ABB RAPID module: Module1.mod

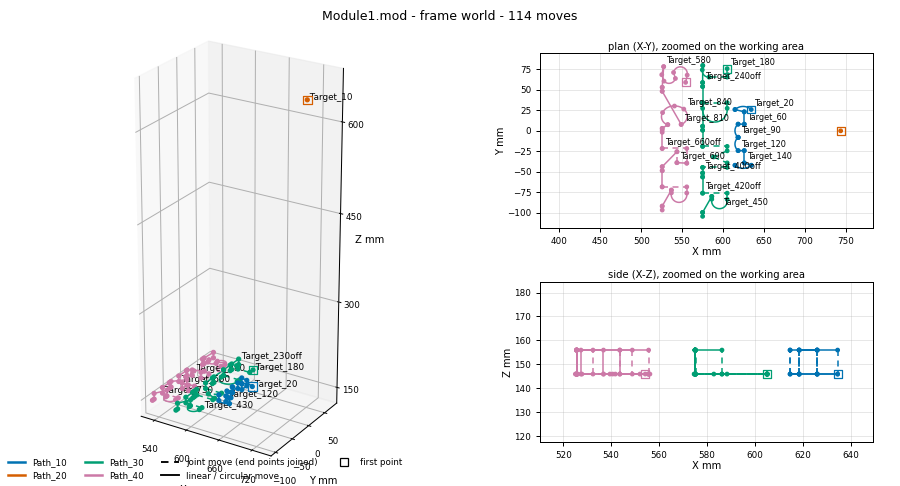
[picture p0: tool path of Module1.mod in frame world, 114 of 114 moves have a stored position in this frame; points joined in program order, loops and branches not executed]
MODULE Module1
    CONST robtarget Target_20:=[[25.588,146.054,0],[1,0,0,0],[0,0,0,1],[9E+09,9E+09,9E+09,9E+09,9E+09,9E+09]];
    CONST robtarget Target_30:=[[35.494,149.81,0],[1,0,0,0],[0,0,0,1],[9E+09,9E+09,9E+09,9E+09,9E+09,9E+09]];
    CONST robtarget Target_Home:=[[306.283094642,150.004,-445.953252285],[1,0,0.000000007,0],[0,0,0,1],[9E+09,9E+09,9E+09,9E+09,9E+09,9E+09]];
    CONST robtarget Target_10:=[[-83.715981405,120.000002402,-514.953287941],[1,-0.000000013,-0.000000023,0.000000007],[-1,0,0,0],[9E+09,9E+09,9E+09,9E+09,9E+09,9E+09]];
    CONST robtarget Target_40:=[[45.401,146.054,0],[1,0,0,0],[0,0,0,1],[9E+09,9E+09,9E+09,9E+09,9E+09,9E+09]];
    CONST robtarget Target_40off:=[[45.401,146.054,-10],[1,0,0,0],[0,0,0,1],[9E+09,9E+09,9E+09,9E+09,9E+09,9E+09]];
    CONST robtarget Target_50:=[[34.121,143.221,0],[1,0,0,0],[0,0,0,1],[9E+09,9E+09,9E+09,9E+09,9E+09,9E+09]];
    CONST robtarget Target_50off:=[[34.121,143.221,-10],[1,0,0,0],[0,0,0,1],[9E+09,9E+09,9E+09,9E+09,9E+09,9E+09]];
    CONST robtarget Target_60:=[[34.121,128.148,0],[1,0,0,0],[0,0,0,1],[9E+09,9E+09,9E+09,9E+09,9E+09,9E+09]];
    CONST robtarget Target_60off:=[[34.121,128.148,-10],[1,0,0,0],[0,0,0,1],[9E+09,9E+09,9E+09,9E+09,9E+09,9E+09]];
    CONST robtarget Target_70:=[[41.621,128.173,0],[1,0,0,0],[0,0,0,1],[9E+09,9E+09,9E+09,9E+09,9E+09,9E+09]];
    CONST robtarget Target_70off:=[[41.621,128.173,-10],[1,0,0,0],[0,0,0,1],[9E+09,9E+09,9E+09,9E+09,9E+09,9E+09]];
    CONST robtarget Target_80:=[[45.462,120.186,0],[1,0,0,0],[0,0,0,1],[9E+09,9E+09,9E+09,9E+09,9E+09,9E+09]];
    CONST robtarget Target_90:=[[41.621,112.188,0],[1,0,0,0],[0,0,0,1],[9E+09,9E+09,9E+09,9E+09,9E+09,9E+09]];
    CONST robtarget Target_90off:=[[41.621,112.188,-10],[1,0,0,0],[0,0,0,1],[9E+09,9E+09,9E+09,9E+09,9E+09,9E+09]];
    CONST robtarget Target_110:=[[45.462,103.801,0],[1,0,0,0],[0,0,0,1],[9E+09,9E+09,9E+09,9E+09,9E+09,9E+09]];
    CONST robtarget Target_110off:=[[45.462,103.801,-10],[1,0,0,0],[0,0,0,1],[9E+09,9E+09,9E+09,9E+09,9E+09,9E+09]];
    CONST robtarget Target_120:=[[41.621,95.802,0],[1,0,0,0],[0,0,0,1],[9E+09,9E+09,9E+09,9E+09,9E+09,9E+09]];
    CONST robtarget Target_120off:=[[41.621,95.802,-10],[1,0,0,0],[0,0,0,1],[9E+09,9E+09,9E+09,9E+09,9E+09,9E+09]];
    CONST robtarget Target_130:=[[34.121,95.839,0],[1,0,0,0],[0,0,0,1],[9E+09,9E+09,9E+09,9E+09,9E+09,9E+09]];
    CONST robtarget Target_130off:=[[34.121,95.839,-10],[1,0,0,0],[0,0,0,1],[9E+09,9E+09,9E+09,9E+09,9E+09,9E+09]];
    CONST robtarget Target_140:=[[34.121,80.766,0],[1,0,0,0],[0,0,0,1],[9E+09,9E+09,9E+09,9E+09,9E+09,9E+09]];
    CONST robtarget Target_140off:=[[34.121,80.766,-10],[1,0,0,0],[0,0,0,1],[9E+09,9E+09,9E+09,9E+09,9E+09,9E+09]];
    CONST robtarget Target_150:=[[25.588,77.934,0],[1,0,0,0],[0,0,0,1],[9E+09,9E+09,9E+09,9E+09,9E+09,9E+09]];
    CONST robtarget Target_150off:=[[25.588,77.934,-10],[1,0,0,0],[0,0,0,1],[9E+09,9E+09,9E+09,9E+09,9E+09,9E+09]];
    CONST robtarget Target_160:=[[35.494,74.178,0],[1,0,0,0],[0,0,0,1],[9E+09,9E+09,9E+09,9E+09,9E+09,9E+09]];
    CONST robtarget Target_170:=[[45.401,77.934,0],[1,0,0,0],[0,0,0,1],[9E+09,9E+09,9E+09,9E+09,9E+09,9E+09]];
    CONST robtarget Target_170off:=[[45.401,77.934,-10],[1,0,0,0],[0,0,0,1],[9E+09,9E+09,9E+09,9E+09,9E+09,9E+09]];
    CONST robtarget Target_100:=[[41.621,111.787,0],[1,0,0,0],[0,0,0,1],[9E+09,9E+09,9E+09,9E+09,9E+09,9E+09]];
    CONST robtarget Target_100off:=[[41.621,111.787,-10],[1,0,0,0],[0,0,0,1],[9E+09,9E+09,9E+09,9E+09,9E+09,9E+09]];
    CONST robtarget Target_180:=[[55,195.989,0],[1,0,0,0],[0,0,0,1],[9E+09,9E+09,9E+09,9E+09,9E+09,9E+09]];
    CONST robtarget Target_190:=[[55,185.656,0],[1,0,0,0],[0,0,0,1],[9E+09,9E+09,9E+09,9E+09,9E+09,9E+09]];
    CONST robtarget Target_200:=[[77.196,185.656,0],[1,0,0,0],[0,0,0,1],[9E+09,9E+09,9E+09,9E+09,9E+09,9E+09]];
    CONST robtarget Target_210:=[[83.274,188.063,0],[1,0,0,0],[0,0,0,1],[9E+09,9E+09,9E+09,9E+09,9E+09,9E+09]];
    CONST robtarget Target_220:=[[85.413,194.53,0],[1,0,0,0],[0,0,0,1],[9E+09,9E+09,9E+09,9E+09,9E+09,9E+09]];
    CONST robtarget Target_230:=[[84.83,199.83,0],[1,0,0,0],[0,0,0,1],[9E+09,9E+09,9E+09,9E+09,9E+09,9E+09]];
    CONST robtarget Target_240:=[[85,178.995,0],[1,0,0,0],[0,0,0,1],[9E+09,9E+09,9E+09,9E+09,9E+09,9E+09]];
    CONST robtarget Target_230off:=[[84.83,199.83,-10],[1,0,0,0],[0,0,0,1],[9E+09,9E+09,9E+09,9E+09,9E+09,9E+09]];
    CONST robtarget Target_240off:=[[85,178.995,-10],[1,0,0,0],[0,0,0,1],[9E+09,9E+09,9E+09,9E+09,9E+09,9E+09]];
    CONST robtarget Target_250:=[[85,174.182,0],[1,0,0,0],[0,0,0,1],[9E+09,9E+09,9E+09,9E+09,9E+09,9E+09]];
    CONST robtarget Target_260:=[[55,154.392,0],[1,0,0,0],[0,0,0,1],[9E+09,9E+09,9E+09,9E+09,9E+09,9E+09]];
    CONST robtarget Target_250off:=[[85,174.182,-10],[1,0,0,0],[0,0,0,1],[9E+09,9E+09,9E+09,9E+09,9E+09,9E+09]];
    CONST robtarget Target_260off:=[[55,154.392,-10],[1,0,0,0],[0,0,0,1],[9E+09,9E+09,9E+09,9E+09,9E+09,9E+09]];
    CONST robtarget Target_270:=[[55,147.561,0],[1,0,0,0],[0,0,0,1],[9E+09,9E+09,9E+09,9E+09,9E+09,9E+09]];
    CONST robtarget Target_280:=[[70.024,130.737,0],[1,0,0,0],[0,0,0,1],[9E+09,9E+09,9E+09,9E+09,9E+09,9E+09]];
    CONST robtarget Target_290:=[[85,147.488,0],[1,0,0,0],[0,0,0,1],[9E+09,9E+09,9E+09,9E+09,9E+09,9E+09]];
    CONST robtarget Target_300:=[[85,154.392,0],[1,0,0,0],[0,0,0,1],[9E+09,9E+09,9E+09,9E+09,9E+09,9E+09]];
    CONST robtarget Target_300off:=[[85,154.392,-10],[1,0,0,0],[0,0,0,1],[9E+09,9E+09,9E+09,9E+09,9E+09,9E+09]];
    CONST robtarget Target_310:=[[85,125.632,0],[1,0,0,0],[0,0,0,1],[9E+09,9E+09,9E+09,9E+09,9E+09,9E+09]];
    CONST robtarget Target_320:=[[85,120.818,0],[1,0,0,0],[0,0,0,1],[9E+09,9E+09,9E+09,9E+09,9E+09,9E+09]];
    CONST robtarget Target_310off:=[[85,125.632,-10],[1,0,0,0],[0,0,0,1],[9E+09,9E+09,9E+09,9E+09,9E+09,9E+09]];
    CONST robtarget Target_320off:=[[85,120.818,-10],[1,0,0,0],[0,0,0,1],[9E+09,9E+09,9E+09,9E+09,9E+09,9E+09]];
    CONST robtarget Target_330:=[[85,101.029,0],[1,0,0,0],[0,0,0,1],[9E+09,9E+09,9E+09,9E+09,9E+09,9E+09]];
    CONST robtarget Target_330off:=[[85,101.029,-10],[1,0,0,0],[0,0,0,1],[9E+09,9E+09,9E+09,9E+09,9E+09,9E+09]];
    CONST robtarget Target_340:=[[55,101.029,0],[1,0,0,0],[0,0,0,1],[9E+09,9E+09,9E+09,9E+09,9E+09,9E+09]];
    CONST robtarget Target_350:=[[55,95.583,0],[1,0,0,0],[0,0,0,1],[9E+09,9E+09,9E+09,9E+09,9E+09,9E+09]];
    CONST robtarget Target_360:=[[71.702,88.096,0],[1,0,0,0],[0,0,0,1],[9E+09,9E+09,9E+09,9E+09,9E+09,9E+09]];
    CONST robtarget Target_370:=[[55,80.851,0],[1,0,0,0],[0,0,0,1],[9E+09,9E+09,9E+09,9E+09,9E+09,9E+09]];
    CONST robtarget Target_380:=[[55,75.308,0],[1,0,0,0],[0,0,0,1],[9E+09,9E+09,9E+09,9E+09,9E+09,9E+09]];
    CONST robtarget Target_390:=[[85,75.308,0],[1,0,0,0],[0,0,0,1],[9E+09,9E+09,9E+09,9E+09,9E+09,9E+09]];
    CONST robtarget Target_390off:=[[85,75.308,-10],[1,0,0,0],[0,0,0,1],[9E+09,9E+09,9E+09,9E+09,9E+09,9E+09]];
    CONST robtarget Target_400:=[[85,68.452,0],[1,0,0,0],[0,0,0,1],[9E+09,9E+09,9E+09,9E+09,9E+09,9E+09]];
    CONST robtarget Target_400off:=[[85,68.452,-10],[1,0,0,0],[0,0,0,1],[9E+09,9E+09,9E+09,9E+09,9E+09,9E+09]];
    CONST robtarget Target_410:=[[85,63.639,0],[1,0,0,0],[0,0,0,1],[9E+09,9E+09,9E+09,9E+09,9E+09,9E+09]];
    CONST robtarget Target_420:=[[85,43.849,0],[1,0,0,0],[0,0,0,1],[9E+09,9E+09,9E+09,9E+09,9E+09,9E+09]];
    CONST robtarget Target_410off:=[[85,63.639,-10],[1,0,0,0],[0,0,0,1],[9E+09,9E+09,9E+09,9E+09,9E+09,9E+09]];
    CONST robtarget Target_420off:=[[85,43.849,-10],[1,0,0,0],[0,0,0,1],[9E+09,9E+09,9E+09,9E+09,9E+09,9E+09]];
    CONST robtarget Target_430:=[[55,43.849,0],[1,0,0,0],[0,0,0,1],[9E+09,9E+09,9E+09,9E+09,9E+09,9E+09]];
    CONST robtarget Target_440:=[[55,36.313,0],[1,0,0,0],[0,0,0,1],[9E+09,9E+09,9E+09,9E+09,9E+09,9E+09]];
    CONST robtarget Target_450:=[[64.044,24.887,0],[1,0,0,0],[0,0,0,1],[9E+09,9E+09,9E+09,9E+09,9E+09,9E+09]];
    CONST robtarget Target_460:=[[73.817,36.483,0],[1,0,0,0],[0,0,0,1],[9E+09,9E+09,9E+09,9E+09,9E+09,9E+09]];
    CONST robtarget Target_470:=[[73.817,39.862,0],[1,0,0,0],[0,0,0,1],[9E+09,9E+09,9E+09,9E+09,9E+09,9E+09]];
    CONST robtarget Target_480:=[[85,20.316,0],[1,0,0,0],[0,0,0,1],[9E+09,9E+09,9E+09,9E+09,9E+09,9E+09]];
    CONST robtarget Target_470off:=[[73.817,39.862,-10],[1,0,0,0],[0,0,0,1],[9E+09,9E+09,9E+09,9E+09,9E+09,9E+09]];
    CONST robtarget Target_480off:=[[85,20.316,-10],[1,0,0,0],[0,0,0,1],[9E+09,9E+09,9E+09,9E+09,9E+09,9E+09]];
    CONST robtarget Target_490:=[[85,15.502,0],[1,0,0,0],[0,0,0,1],[9E+09,9E+09,9E+09,9E+09,9E+09,9E+09]];
    CONST robtarget Target_500:=[[105.804,179.214,0],[1,0,0,0],[0,0,0,1],[9E+09,9E+09,9E+09,9E+09,9E+09,9E+09]];
    CONST robtarget Target_510:=[[103.859,188.136,0],[1,0,0,0],[0,0,0,1],[9E+09,9E+09,9E+09,9E+09,9E+09,9E+09]];
    CONST robtarget Target_520:=[[112.441,198.225,0],[1,0,0,0],[0,0,0,1],[9E+09,9E+09,9E+09,9E+09,9E+09,9E+09]];
    CONST robtarget Target_530:=[[120.513,191.321,0],[1,0,0,0],[0,0,0,1],[9E+09,9E+09,9E+09,9E+09,9E+09,9E+09]];
    CONST robtarget Target_540:=[[118.276,184.003,0],[1,0,0,0],[0,0,0,1],[9E+09,9E+09,9E+09,9E+09,9E+09,9E+09]];
    CONST robtarget Target_550:=[[125.837,178.047,0],[1,0,0,0],[0,0,0,1],[9E+09,9E+09,9E+09,9E+09,9E+09,9E+09]];
    CONST robtarget Target_560:=[[132.206,180.77,0],[1,0,0,0],[0,0,0,1],[9E+09,9E+09,9E+09,9E+09,9E+09,9E+09]];
    CONST robtarget Target_550off:=[[125.837,178.047,-10],[1,0,0,0],[0,0,0,1],[9E+09,9E+09,9E+09,9E+09,9E+09,9E+09]];
    CONST robtarget Target_560off:=[[132.206,180.77,-10],[1,0,0,0],[0,0,0,1],[9E+09,9E+09,9E+09,9E+09,9E+09,9E+09]];
    CONST robtarget Target_570:=[[134.929,188.598,0],[1,0,0,0],[0,0,0,1],[9E+09,9E+09,9E+09,9E+09,9E+09,9E+09]];
    CONST robtarget Target_580:=[[132.595,198.444,0],[1,0,0,0],[0,0,0,1],[9E+09,9E+09,9E+09,9E+09,9E+09,9E+09]];
    CONST robtarget Target_590:=[[134.394,173.209,0],[1,0,0,0],[0,0,0,1],[9E+09,9E+09,9E+09,9E+09,9E+09,9E+09]];
    CONST robtarget Target_600:=[[134.394,168.395,0],[1,0,0,0],[0,0,0,1],[9E+09,9E+09,9E+09,9E+09,9E+09,9E+09]];
    CONST robtarget Target_610:=[[106.388,127.553,0],[1,0,0,0],[0,0,0,1],[9E+09,9E+09,9E+09,9E+09,9E+09,9E+09]];
    CONST robtarget Target_580off:=[[132.595,198.444,-10],[1,0,0,0],[0,0,0,1],[9E+09,9E+09,9E+09,9E+09,9E+09,9E+09]];
    CONST robtarget Target_590off:=[[134.394,173.209,-10],[1,0,0,0],[0,0,0,1],[9E+09,9E+09,9E+09,9E+09,9E+09,9E+09]];
    CONST robtarget Target_600off:=[[134.394,168.395,-10],[1,0,0,0],[0,0,0,1],[9E+09,9E+09,9E+09,9E+09,9E+09,9E+09]];
    CONST robtarget Target_610off:=[[106.388,127.553,-10],[1,0,0,0],[0,0,0,1],[9E+09,9E+09,9E+09,9E+09,9E+09,9E+09]];
    CONST robtarget Target_620:=[[119.419,150.308,0],[1,0,0,0],[0,0,0,1],[9E+09,9E+09,9E+09,9E+09,9E+09,9E+09]];
    CONST robtarget Target_630:=[[132.352,127.553,0],[1,0,0,0],[0,0,0,1],[9E+09,9E+09,9E+09,9E+09,9E+09,9E+09]];
    CONST robtarget Target_640:=[[134.394,123.055,0],[1,0,0,0],[0,0,0,1],[9E+09,9E+09,9E+09,9E+09,9E+09,9E+09]];
    CONST robtarget Target_630off:=[[132.352,127.553,-10],[1,0,0,0],[0,0,0,1],[9E+09,9E+09,9E+09,9E+09,9E+09,9E+09]];
    CONST robtarget Target_640off:=[[134.394,123.055,-10],[1,0,0,0],[0,0,0,1],[9E+09,9E+09,9E+09,9E+09,9E+09,9E+09]];
    CONST robtarget Target_650:=[[134.394,118.241,0],[1,0,0,0],[0,0,0,1],[9E+09,9E+09,9E+09,9E+09,9E+09,9E+09]];
    CONST robtarget Target_660:=[[134.394,98.452,0],[1,0,0,0],[0,0,0,1],[9E+09,9E+09,9E+09,9E+09,9E+09,9E+09]];
    CONST robtarget Target_650off:=[[134.394,120.939,-10],[1,0,0,0],[0,0,0,1],[9E+09,9E+09,9E+09,9E+09,9E+09,9E+09]];
    CONST robtarget Target_660off:=[[134.394,98.452,-10],[1,0,0,0],[0,0,0,1],[9E+09,9E+09,9E+09,9E+09,9E+09,9E+09]];
    CONST robtarget Target_670:=[[104.394,98.452,0],[1,0,0,0],[0,0,0,1],[9E+09,9E+09,9E+09,9E+09,9E+09,9E+09]];
    CONST robtarget Target_680:=[[104.394,80.511,0],[1,0,0,0],[0,0,0,1],[9E+09,9E+09,9E+09,9E+09,9E+09,9E+09]];
    CONST robtarget Target_690:=[[116.404,81.094,0],[1,0,0,0],[0,0,0,1],[9E+09,9E+09,9E+09,9E+09,9E+09,9E+09]];
    CONST robtarget Target_680off:=[[104.394,80.511,-10],[1,0,0,0],[0,0,0,1],[9E+09,9E+09,9E+09,9E+09,9E+09,9E+09]];
    CONST robtarget Target_690off:=[[116.404,81.094,-10],[1,0,0,0],[0,0,0,1],[9E+09,9E+09,9E+09,9E+09,9E+09,9E+09]];
    CONST robtarget Target_700:=[[116.404,94.465,0],[1,0,0,0],[0,0,0,1],[9E+09,9E+09,9E+09,9E+09,9E+09,9E+09]];
    CONST robtarget Target_710:=[[134.394,76.159,0],[1,0,0,0],[0,0,0,1],[9E+09,9E+09,9E+09,9E+09,9E+09,9E+09]];
    CONST robtarget Target_700off:=[[116.404,94.465,-10],[1,0,0,0],[0,0,0,1],[9E+09,9E+09,9E+09,9E+09,9E+09,9E+09]];
    CONST robtarget Target_710off:=[[134.394,76.159,-10],[1,0,0,0],[0,0,0,1],[9E+09,9E+09,9E+09,9E+09,9E+09,9E+09]];
    CONST robtarget Target_720:=[[134.394,71.345,0],[1,0,0,0],[0,0,0,1],[9E+09,9E+09,9E+09,9E+09,9E+09,9E+09]];
    CONST robtarget Target_730:=[[134.394,51.556,0],[1,0,0,0],[0,0,0,1],[9E+09,9E+09,9E+09,9E+09,9E+09,9E+09]];
    CONST robtarget Target_720off:=[[134.394,71.345,-10],[1,0,0,0],[0,0,0,1],[9E+09,9E+09,9E+09,9E+09,9E+09,9E+09]];
    CONST robtarget Target_730off:=[[134.394,51.556,-10],[1,0,0,0],[0,0,0,1],[9E+09,9E+09,9E+09,9E+09,9E+09,9E+09]];
    CONST robtarget Target_740:=[[104.394,51.556,0],[1,0,0,0],[0,0,0,1],[9E+09,9E+09,9E+09,9E+09,9E+09,9E+09]];
    CONST robtarget Target_750:=[[104.394,44.019,0],[1,0,0,0],[0,0,0,1],[9E+09,9E+09,9E+09,9E+09,9E+09,9E+09]];
    CONST robtarget Target_760:=[[113.438,32.593,0],[1,0,0,0],[0,0,0,1],[9E+09,9E+09,9E+09,9E+09,9E+09,9E+09]];
    CONST robtarget Target_770:=[[123.211,44.19,0],[1,0,0,0],[0,0,0,1],[9E+09,9E+09,9E+09,9E+09,9E+09,9E+09]];
    CONST robtarget Target_780:=[[123.211,47.569,0],[1,0,0,0],[0,0,0,1],[9E+09,9E+09,9E+09,9E+09,9E+09,9E+09]];
    CONST robtarget Target_790:=[[134.394,28.023,0],[1,0,0,0],[0,0,0,1],[9E+09,9E+09,9E+09,9E+09,9E+09,9E+09]];
    CONST robtarget Target_780off:=[[123.211,47.569,-10],[1,0,0,0],[0,0,0,1],[9E+09,9E+09,9E+09,9E+09,9E+09,9E+09]];
    CONST robtarget Target_790off:=[[134.394,28.023,-10],[1,0,0,0],[0,0,0,1],[9E+09,9E+09,9E+09,9E+09,9E+09,9E+09]];
    CONST robtarget Target_800:=[[134.394,23.209,0],[1,0,0,0],[0,0,0,1],[9E+09,9E+09,9E+09,9E+09,9E+09,9E+09]];
    CONST robtarget Target_810:=[[111.201,127.869,0],[1,0,0,0],[0,0,0,1],[9E+09,9E+09,9E+09,9E+09,9E+09,9E+09]];
    CONST robtarget Target_820:=[[127.587,127.553,0],[1,0,0,0],[0,0,0,1],[9E+09,9E+09,9E+09,9E+09,9E+09,9E+09]];
    CONST robtarget Target_810off:=[[111.201,127.869,-10],[1,0,0,0],[0,0,0,1],[9E+09,9E+09,9E+09,9E+09,9E+09,9E+09]];
    CONST robtarget Target_820off:=[[127.587,127.553,-10],[1,0,0,0],[0,0,0,1],[9E+09,9E+09,9E+09,9E+09,9E+09,9E+09]];
    CONST robtarget Target_830:=[[103.859,136.815,0],[1,0,0,0],[0,0,0,1],[9E+09,9E+09,9E+09,9E+09,9E+09,9E+09]];
    CONST robtarget Target_840:=[[107.992,146.564,0],[1,0,0,0],[0,0,0,1],[9E+09,9E+09,9E+09,9E+09,9E+09,9E+09]];
    CONST robtarget Target_850:=[[112.855,149.348,0],[1,0,0,0],[0,0,0,1],[9E+09,9E+09,9E+09,9E+09,9E+09,9E+09]];
    CONST robtarget Target_860:=[[119.419,150.308,0],[1,0,0,0],[0,0,0,1],[9E+09,9E+09,9E+09,9E+09,9E+09,9E+09]];
    CONST robtarget Target_870:=[[126.128,149.323,0],[1,0,0,0],[0,0,0,1],[9E+09,9E+09,9E+09,9E+09,9E+09,9E+09]];
    CONST robtarget Target_880:=[[133.944,142.273,0],[1,0,0,0],[0,0,0,1],[9E+09,9E+09,9E+09,9E+09,9E+09,9E+09]];
    CONST robtarget Target_890:=[[134.71,133.971,0],[1,0,0,0],[0,0,0,1],[9E+09,9E+09,9E+09,9E+09,9E+09,9E+09]];
    PERS tooldata MyNewTool:=[TRUE,[[80.603,0,147.485],[0.866025404,0,0.5,0]],[1,[0,0,1],[1,0,0,0],0,0,0]];
    TASK PERS wobjdata Workobject_2:=[FALSE,TRUE,"",[[0,0,0],[1,0,0,0]],[[660,-120,146],[0,0,1,0]]];
    TASK PERS wobjdata Workobject_1:=[FALSE,TRUE,"",[[0,0,0],[1,0,0,0]],[[749.999,-150.004,90],[0,0,1,0]]];

    PROC main()
        Path_20;
        WaitTime 4;
        Path_10;
        Path_20;
        Path_30;
        Path_20;
        Path_40;
        Path_20;
    ENDPROC
    PROC Path_10()                  !Emoji
        MoveJ Target_20,v100,z10,MyNewTool\WObj:=Workobject_2;
        MoveC Target_30, Target_40, v100,z10,MyNewTool\WObj:=Workobject_2;
        WaitTime 1;
        MoveJ Target_40off,v100,z10,MyNewTool\WObj:=Workobject_2;
        MoveL Target_50off,v100,z10,MyNewTool\WObj:=Workobject_2;
        WaitTime 1;
        MoveJ Target_50,v100,z10,MyNewTool\WObj:=Workobject_2;
        MoveL Target_60,v100,z10,MyNewTool\WObj:=Workobject_2;
        WaitTime 1;
        MoveJ Target_60off,v100,z10,MyNewTool\WObj:=Workobject_2;
        MoveL Target_70off,v100,z10,MyNewTool\WObj:=Workobject_2;
        MoveJ Target_70,v100,z10,MyNewTool\WObj:=Workobject_2;
        WaitTime 1;
        MoveC Target_80,Target_90,v100,z10,MyNewTool\WObj:=Workobject_2;
        MoveJ Target_90off,v100,z10,MyNewTool\WObj:=Workobject_2;
        MoveL Target_100off,v100,z10,MyNewTool\WObj:=Workobject_2;
        MoveJ Target_100,v100,z10,MyNewTool\WObj:=Workobject_2;
        WaitTime 1;
        MoveC Target_110,Target_120,v100,z10,MyNewTool\WObj:=Workobject_2;
        MoveJ Target_120off,v100,z100,MyNewTool\WObj:=Workobject_2;
        MoveL Target_130off,v100,z10,MyNewTool\WObj:=Workobject_2;
        MoveJ Target_130,v100,z10,MyNewTool\WObj:=Workobject_2;
        WaitTime 1;
        MoveL Target_140,v100,z10,MyNewTool\WObj:=Workobject_2;
        MoveJ Target_140off,v100,z10,MyNewTool\WObj:=Workobject_2;
        MoveL Target_150off,v100,z10,MyNewTool\WObj:=Workobject_2;
        MoveJ Target_150,v100,z10,MyNewTool\WObj:=Workobject_2;
        MoveC Target_160,Target_170,v100,z10,MyNewTool\WObj:=Workobject_2;
        WaitTime 1;
        MoveJ Target_170off,v100,z10,MyNewTool\WObj:=Workobject_2;
    ENDPROC
    PROC Path_20() !Home
        MoveJ Target_10,v100,z10,MyNewTool\WObj:=Workobject_2;
    ENDPROC
    PROC Path_30() !Iniciales JDMP
        MoveJ Target_180,v100,z10,MyNewTool\WObj:=Workobject_2;    !J
        MoveJ Target_190,v100,z10,MyNewTool\WObj:=Workobject_2;
        MoveJ Target_200,v100,z10,MyNewTool\WObj:=Workobject_2;
        MoveC Target_210,Target_220,v100,z10,MyNewTool\WObj:=Workobject_2;
        MoveJ Target_230,v100,z10,MyNewTool\WObj:=Workobject_2;
        MoveJ Target_230off,v100,z10,MyNewTool\WObj:=Workobject_2;
        MoveL Target_240off,v100,z10,MyNewTool\WObj:=Workobject_2;
        MoveJ Target_240,v100,z10,MyNewTool\WObj:=Workobject_2;
        MoveJ Target_250,v100,z10,MyNewTool\WObj:=Workobject_2;
        MoveJ Target_250off,v100,z10,MyNewTool\WObj:=Workobject_2;
        MoveL Target_300off,v100,z10,MyNewTool\WObj:=Workobject_2; !D
        MoveL Target_300,v100,z10,MyNewTool\WObj:=Workobject_2;
        MoveJ Target_260,v100,z10,MyNewTool\WObj:=Workobject_2;
        MoveL Target_270,v100,z10,MyNewTool\WObj:=Workobject_2;
        MoveC Target_280,Target_290,v100,z10,MyNewTool\WObj:=Workobject_2;
        MoveJ Target_300,v100,z10,MyNewTool\WObj:=Workobject_2;
        MoveL Target_300off,v100,z10,MyNewTool\WObj:=Workobject_2;
        MoveL Target_310off,v100,z10,MyNewTool\WObj:=Workobject_2;
        MoveJ Target_310,v100,z10,MyNewTool\WObj:=Workobject_2;
        MoveJ Target_320,v100,z10,MyNewTool\WObj:=Workobject_2;
        MoveL Target_320off,v100,z10,MyNewTool\WObj:=Workobject_2;
        MoveL Target_330off,v100,z10,MyNewTool\WObj:=Workobject_2; !M
        MoveJ Target_330,v100,z10,MyNewTool\WObj:=Workobject_2;
        MoveJ Target_340,v100,z10,MyNewTool\WObj:=Workobject_2;
        MoveJ Target_350,v100,z10,MyNewTool\WObj:=Workobject_2;
        MoveJ Target_360,v100,z10,MyNewTool\WObj:=Workobject_2;
        MoveJ Target_370,v100,z10,MyNewTool\WObj:=Workobject_2;
        MoveJ Target_380,v100,z10,MyNewTool\WObj:=Workobject_2;
        MoveJ Target_390,v100,z10,MyNewTool\WObj:=Workobject_2;
        MoveJ Target_390off,v100,z10,MyNewTool\WObj:=Workobject_2;
        MoveL Target_400off,v100,z10,MyNewTool\WObj:=Workobject_2;
        MoveJ Target_400,v100,z10,MyNewTool\WObj:=Workobject_2;
        MoveJ Target_410,v100,z10,MyNewTool\WObj:=Workobject_2;
        MoveJ Target_410off,v100,z10,MyNewTool\WObj:=Workobject_2;
        MoveL Target_420off,v100,z10,MyNewTool\WObj:=Workobject_2;
        MoveJ Target_420,v100,z10,MyNewTool\WObj:=Workobject_2;
        MoveJ Target_430,v100,z10,MyNewTool\WObj:=Workobject_2;
        MoveJ Target_440,v100,z10,MyNewTool\WObj:=Workobject_2;
        MoveC Target_450,Target_460,v100,z10,MyNewTool\WObj:=Workobject_2;
        MoveJ Target_470,v100,z10,MyNewTool\WObj:=Workobject_2;
        MoveJ Target_470off,v100,z10,MyNewTool\WObj:=Workobject_2;
        MoveL Target_480off,v100,z10,MyNewTool\WObj:=Workobject_2;
        MoveJ Target_480,v100,z10,MyNewTool\WObj:=Workobject_2;
        MoveJ Target_490,v100,z10,MyNewTool\WObj:=Workobject_2;
    ENDPROC
    PROC Path_40() !Iniciales SCFP
        MoveJ Target_500,v100,z10,MyNewTool\WObj:=Workobject_2;     !S
        MoveL Target_510,v100,z10,MyNewTool\WObj:=Workobject_2;
        MoveC Target_520,Target_530,v100,z10,MyNewTool\WObj:=Workobject_2;
        MoveL Target_540,v100,z100,MyNewTool\WObj:=Workobject_2;
        MoveC Target_550,Target_560,v100,z10,MyNewTool\WObj:=Workobject_2;
        MoveL Target_570,v100,z10,MyNewTool\WObj:=Workobject_2;
        MoveJ Target_580,v100,z10,MyNewTool\WObj:=Workobject_2;
        MoveL Target_580off,v100,z10,MyNewTool\WObj:=Workobject_2;
        MoveL Target_590off,v100,z10,MyNewTool\WObj:=Workobject_2;
        MoveJ Target_590,v100,z10,MyNewTool\WObj:=Workobject_2;
        MoveJ Target_600,v100,z10,MyNewTool\WObj:=Workobject_2;
        MoveL Target_600off,v100,z10,MyNewTool\WObj:=Workobject_2;
        MoveL Target_810off,v100,z10,MyNewTool\WObj:=Workobject_2;  !C
        MoveJ Target_810,v100,z10,MyNewTool\WObj:=Workobject_2;
        MoveC Target_830,Target_840,v100,z10,MyNewTool\WObj:=Workobject_2;
        MoveC Target_850,Target_860,v100,z10,MyNewTool\WObj:=Workobject_2;
        MoveC Target_870,Target_880,v100,z10,MyNewTool\WObj:=Workobject_2;
        MoveC Target_890,Target_820,v100,z10,MyNewTool\WObj:=Workobject_2;
        MoveJ Target_820off,v100,z10,MyNewTool\WObj:=Workobject_2;
        MoveJ Target_640off,v100,z10,MyNewTool\WObj:=Workobject_2;  !F
        MoveJ Target_640,v100,z10,MyNewTool\WObj:=Workobject_2;
        MoveJ Target_650,v100,z10,MyNewTool\WObj:=Workobject_2;
        MoveL Target_650off,v100,z10,MyNewTool\WObj:=Workobject_2;
        MoveL Target_660off,v100,z10,MyNewTool\WObj:=Workobject_2;
        MoveJ Target_660,v100,z10,MyNewTool\WObj:=Workobject_2;
        MoveJ Target_670,v100,z10,MyNewTool\WObj:=Workobject_2;
        MoveJ Target_680,v100,z10,MyNewTool\WObj:=Workobject_2;
        MoveJ Target_680off,v100,z10,MyNewTool\WObj:=Workobject_2;
        MoveL Target_690off,v100,z10,MyNewTool\WObj:=Workobject_2;
        MoveJ Target_690,v100,z10,MyNewTool\WObj:=Workobject_2;
        MoveJ Target_700,v100,z10,MyNewTool\WObj:=Workobject_2;
        MoveL Target_700off,v100,z10,MyNewTool\WObj:=Workobject_2;
        MoveL Target_710off,v100,z10,MyNewTool\WObj:=Workobject_2;
        MoveJ Target_710,v100,z10,MyNewTool\WObj:=Workobject_2;
        MoveJ Target_720,v100,z10,MyNewTool\WObj:=Workobject_2;
        MoveL Target_720off,v100,z10,MyNewTool\WObj:=Workobject_2;
        MoveL Target_730off,v100,z10,MyNewTool\WObj:=Workobject_2;
        MoveJ Target_730,v100,z10,MyNewTool\WObj:=Workobject_2;
        MoveJ Target_740,v100,z10,MyNewTool\WObj:=Workobject_2;
        MoveJ Target_750,v100,z10,MyNewTool\WObj:=Workobject_2;
        MoveC Target_760,Target_770,v100,z10,MyNewTool\WObj:=Workobject_2;
        MoveJ Target_780,v100,z10,MyNewTool\WObj:=Workobject_2;
        MoveL Target_780off,v100,z10,MyNewTool\WObj:=Workobject_2;
        MoveL Target_790off,v100,z10,MyNewTool\WObj:=Workobject_2;
        MoveJ Target_790,v100,z10,MyNewTool\WObj:=Workobject_2;
        MoveL Target_800,v100,z10,MyNewTool\WObj:=Workobject_2;
    ENDPROC
ENDMODULE
